FUNCTION F_CopyMem : UDINT
VAR_INPUT
    Source      : ANY;
    Destination : ANY;
END_VAR
VAR
END_VAR

IF Destination.diSize = Source.diSize THEN
    memcpy(destAddr := Destination.pValue,
           srcAddr  := Source.pValue,
           n        := F_DINT_TO_UDINT(Source.diSize));
END_IF

END_FUNCTION

(* stored: Version 1.1.0.1, ProductVersion 3.1.4024.12
   POU F_CopyMem: Id {acfda558-155a-4b88-8f3a-a5ac87315fb0}, SpecialFunc None *)
